Fanuc KAREL source: kt00785.KL

-- PROVISIONAL review KL for V1013-1; original PC SHA256 59fac55b7c46743da327756d05d724b68f35116e897c54bef7bb790eaaeb7aed
-- Incomplete behavior may be omitted. Consult companion uncertainty JSON. Do not deploy.
PROGRAM KT00785
%NOLOCKGROUP
VAR
  I1 : INTEGER
  I2 : INTEGER
  OUT : REAL
BEGIN
  -- UNRESOLVED_PC offsets 5-16; opcodes 2E,23
  -- UNRESOLVED_PC offsets 21-32; opcodes 2E,23
  -- UNRESOLVED_PC offsets 37-48; opcodes 2E,23
  -- UNRESOLVED_PC offsets 53-64; opcodes 2E,23
  -- UNRESOLVED_PC offsets 69-86; opcodes 27,27,21,64,76,23
  -- UNRESOLVED_PC offsets 91-95; opcodes 7F
END KT00785
